//Anche FB2 Implementa l'interfaccia iFB
//Posso considerarla come un'altra implementazione della stessa

FUNCTION_BLOCK PUBLIC FB2 IMPLEMENTS iFb
VAR_INPUT
END_VAR
VAR_OUTPUT
END_VAR
VAR
	fInternalInput1 : REAL;
	fInternalInput2 : REAL;
END_VAR

{warning 'add property implementation'}
PROPERTY fInput1 : REAL
GET
fInput1 := this^.fInternalInput1;
END_GET
SET
this^.fInternalInput1 := fInput1;
END_SET
END_PROPERTY

{warning 'add property implementation'}
PROPERTY fInput2 : REAL
GET
fInput2 := this^.fInternalInput2;
END_GET
SET
this^.fInternalInput2 := fInput2;
END_SET
END_PROPERTY

{warning 'add method implementation'}
METHOD returnValue : REAL
//Implementazione Interfaccia con moltiplicazione
returnValue := this^.fInput1 * this^.fInput2;
END_METHOD

END_FUNCTION_BLOCK

(* stored: Version 1.1.0.1, ProductVersion 3.1.4022.16
   POU FB2: Id {413a6a38-7614-4c1d-aeab-92753ab51c6e}, SpecialFunc None
   Property fInput1: Id {ffa9bc79-1456-46dc-94a0-ec5167f9f9b0}
   Get Get: Id {9a67498a-b28e-4503-b65c-6c7eaf36de2a}
   Set Set: Id {6a39df0c-cd8e-4c69-a7a6-872357a36c70}
   Property fInput2: Id {62a3d6e3-2695-4ab8-8f48-17b0d403e21a}
   Get Get: Id {b7615b87-26fd-4270-abfa-c7714cdd9fbe}
   Set Set: Id {eefeb826-7d41-49b8-9ad8-df5012f99532}
   Method returnValue: Id {4b95e94b-8f6d-4b5e-a7ad-acf679323fd0} *)
